{attribute 'linkalways'} 
{attribute 'no_explicit_call' := 'This FB is a CLASS and must be accessed using methods or properties'}
{attribute 'enable_dynamic_creation'}
FUNCTION_BLOCK FINAL MODABS_LREAL EXTENDS Node
VAR
	value : _LREAL(0.0);
	arg : _LREAL(0.0);
	out : _LREAL(0.0);
END_VAR

METHOD PUBLIC Clone : I_Node
VAR
	pNode : POINTER TO MODABS_LREAL;
END_VAR
pNode := __NEW(MODABS_LREAL);
Clone := pNode^;
END_METHOD

METHOD FB_init : BOOL
VAR_INPUT
	bInitRetains : BOOL; // if TRUE, the retain variables are initialized (warm start / cold start)
	bInCopyCode : BOOL;  // if TRUE, the instance afterwards gets moved into the copy code (online change)
END_VAR
AddInput('value',THIS^.value);
AddInput('arg',THIS^.arg);
AddOutput('out', THIS^.out);
END_METHOD

METHOD PROTECTED OnExecute
VAR
END_VAR
out.Value := MODABS(value.Value, arg.Value);
END_METHOD

END_FUNCTION_BLOCK

(* stored: Version 1.1.0.1, ProductVersion 3.1.4024.15
   POU MODABS_LREAL: Id {15c53ca2-b091-4084-bd8e-96a2a88ee03f}, SpecialFunc None
   Folder Constructor: Id {738cad8d-bf74-4110-8bca-f3c97dc02a5b}
   Method Clone: Id {f7779b04-6fcb-4af6-b947-fc0d28046c18}
   Method FB_init: Id {af6a19b7-fe44-4533-8463-fb0ccf965cba}
   Method OnExecute: Id {84b6b207-1dff-40f8-b1ba-dc9a90eef560} *)
